INTERFACE I_Syntax_Widget EXTENDS __System.IQueryInterface

METHOD M_GetValue : INT
END_METHOD

METHOD M_Init : BOOL
END_METHOD

PROPERTY P_Name : STRING
GET
END_GET
END_PROPERTY

END_INTERFACE

(* stored: Version 1.1.0.1, ProductVersion 3.1.4024.16
   Itf I_Syntax_Widget: Id {82848a68-ef61-408e-ac30-65608590b957}
   Method M_GetValue: Id {78409f0b-e366-4d15-9455-6f500c60c8d8}
   Method M_Init: Id {5899f78d-24ab-4969-b34b-894490a47980}
   Property P_Name: Id {2154926d-de2c-40ee-a734-5322b86599f2}
   Get Get: Id {53c63b8c-93ba-46e3-aa7b-f567464634ad} *)
